FUNCTION_BLOCK EL3152
VAR
	_io : EL3xx2_Data;
	{attribute addProperty Name "WcState"}
	_wcState : WcStateInputToggle;
	{attribute addProperty Name "Info data"}
	_infoData : InfoDataAds;
END_VAR

PROPERTY IO : REFERENCE TO EL3xx2_Data
GET
IO REF= _io;
END_GET
END_PROPERTY

PROPERTY WcState : REFERENCE TO WcStateInputToggle
GET
WcState REF= _wcState;
END_GET
END_PROPERTY

END_FUNCTION_BLOCK

(* stored: Version 1.1.0.1, ProductVersion 3.1.4024.9
   POU EL3152: Id {1d58b435-d1ca-0874-14ed-5313c2ea7eec}, SpecialFunc None
   Property IO: Id {631db380-9bb2-0fd7-08a1-2fed60b3a93e}
   Get Get: Id {5db5f6b6-f501-02a5-077c-bedece84dda0}
   Property WcState: Id {156ea18e-4a90-0f28-2248-274e17c83cb2}
   Get Get: Id {cdbab142-48d4-0db3-127d-c245e44afe60} *)
